TYPE ST_SEW_Movisafe_CSSx1a_Config :
STRUCT	
	bForceMode			: BOOL; //Ignore process data from fieldbus.
	bSwapProcessData	: BOOL; //Reverse process data byte order from/to fieldbus.
END_STRUCT
END_TYPE

(* stored: Version 1.1.0.1, ProductVersion 3.1.4024.12
   DUT ST_SEW_Movisafe_CSSx1a_Config: Id {8511d0ac-9b64-0794-3fcf-731ce4a07f75} *)
